(* CoDeSys 2.3 export: plc_sample.exp *)

(* POU MAIN, ST *)
PROGRAM MAIN
VAR
	StartTest: BOOL;
	StopTest: BOOL;
	TestIsRunning: BOOL;
END_VAR
IF StartTest THEN
	StartTest := FALSE;
	TestIsRunning := TRUE;
END_IF

IF StopTest THEN
	StopTest := FALSE;
	TestIsRunning := FALSE;
END_IF
END_PROGRAM
